Staubli VAL3: updateJointVelocityControl.pgx

program updateJointVelocityControl(RobotState& x_robotState, RobotCommand& x_robotCommand, bool& x_bError, bool b_isFirstCall)
begin
  // Copyright 2025 ICUBE Laboratory, University of Strasbourg
  //
  // Licensed under the Apache License, Version 2.0 (the "License");
  // you may not use this file except in compliance with the License.
  // You may obtain a copy of the License at
  //
  //     http://www.apache.org/licenses/LICENSE-2.0
  //
  // Unless required by applicable law or agreed to in writing, software
  // distributed under the License is distributed on an "AS IS" BASIS,
  // WITHOUT WARRANTIES OR CONDITIONS OF ANY KIND, either express or implied.
  // See the License for the specific language governing permissions and
  // limitations under the License.

  if (!x_robotState.bMotionPossible)
      logMsg("ros2_server::jointVelocityControl : motion not possible, aborting...", 2)
      call stopJointVelocityControl(x_bError)
      x_bError = true
      return
  endIf

  // Check command is valid
  if (!x_robotCommand.bIsValid)
      logMsg("ros2_server::jointVelocityControl : invalid command, aborting...", 2)
      call stopJointVelocityControl(x_bError)
      x_bError = true
      return
  endIf

  if (x_robotCommand.nMotionCmdType != 3)
      logMsg("ros2_server::jointVelocityControl : unexpected command type, aborting...", 2)
      call stopJointVelocityControl(x_bError)
      x_bError = true
      return
  endIf

  // First call: config motion parameters
  if(b_isFirstCall == true)
    resetMotion()
    // Set velocity control parameters
    // $velJoint(motionCfgVel.tTool, motionCfgVel.mMaxSpeed)
  endIf

  // Check safety limits
  // TODO


  // Execute velocity motion command
  // $setVelCmd(x_robotCommand.nMotionCmdData)
  logMsg("ros2_server::jointVelocityControl : not yet implemented", 1)
  x_bError = true
  return

  // OK
  x_bError = false
end
